FUNCTION F_SetWarning : BOOL
VAR_INPUT
	nWrningID	: INT;
	nLine		: INT;
END_VAR
VAR
END_VAR

IF nLine = 1 THEN
	bWarning  := TRUE;
ELSIF nLine = 2 THEN
	bWarning2 := TRUE;
END_IF
nWarningID	:= nWrningID;

END_FUNCTION

(* stored: Version 1.1.0.1, ProductVersion 3.1.4024.12
   POU F_SetWarning: Id {2b26f2d5-d0c6-429d-803a-56a467e14430}, SpecialFunc None *)
